FUNCTION_BLOCK FB_SendDriveReset_Left
VAR_INPUT
	DriveReset : BOOL;
END_VAR
VAR_OUTPUT
END_VAR
VAR
	TxMessage : EXTCANQUEUE;
END_VAR
VAR_IN_OUT
	CAN_OUTPUTS_Left : CANTXQUEUESTRUCT_E_32;
	CAN_INPUTS_Left : CANRXQUEUESTRUCT_E_32;
END_VAR


TxMessage.cobId := 150;
TxMessage.length := 1;
TxMessage.data[0] :=  BOOL_TO_BYTE(DriveReset);
CAN_OUTPUTS_Left.TxMessages[9] := TxMessage;
//CAN_OUTPUTS.NoOfTxMessages := 1;

END_FUNCTION_BLOCK

(* stored: Version 1.1.0.1
   POU FB_SendDriveReset_Left: Id {d43fc5b7-a1a3-4570-bd9a-76a1b8f88161}, SpecialFunc None *)
